PROGRAM MAIN
VAR
END_VAR

END_PROGRAM

(* stored: Version 1.1.0.1
   POU MAIN: Id {075e54ac-c372-45bb-bd99-d8cf5a03bf2f} *)
